TYPE ST_OpenLoopSettings :
STRUCT
	fBoreArea : LREAL := 0.0033183;
	fAnnulusArea : LREAL := 0.0023562;
END_STRUCT
END_TYPE

(* stored: Version 1.1.0.1, ProductVersion 3.1.4024.12
   DUT ST_OpenLoopSettings: Id {8500dbef-7f7e-4976-9606-7ef1170dfe1c} *)
